Universal Robots PolyScope program: demo07_client_server.urp

Program demo07_client_server (installation=bbl_01 directory=/programs createdIn=5.7.0.90932 lastSavedIn=5.7.0.90932 robotSerialNumber=20205300236)
Calibrated DH parameters: a=[-0.000056, -0.241378, -0.055128, 0.000067, -0.000138, 0]; d=[0.151803, -14.462882, 131.163662, -116.569967, 0.085381, 0.091498]; alpha=[1.571556, -0.002127, 0.001765, 1.572165, -1.572257, 0]; deltaTheta=[0, 0.126747, 1.182538, -1.309285, 0, -0.000001]
BeforeStart
  Script: socket_close()
  Wait Sleep waitTime=0.25
  socket_is_open := False
  command_index := 0
Robot Program (runOnlyOnce=false)
  command_index := command_index+1
  Loop While (checkContinuously=false) expression=socket_is_open ≟  False
    socket_is_open := socket_open("192.168.1.1", 30000)
    Wait Sleep waitTime=0.5
  command := socket_read_ascii_float(5)
  response := "Unknown command"
  If command[0]≟5
    Switch expression=command[1]
      Case (caseValue=1)
        MoveL speed 250 mm/s, acceleration 1200 mm/s^2 (useActiveTCP=true) feature=Base
          Waypoint up_pose: TCP in base x=-233.309 y=250.262 z=151.642 mm, rx=0 ry=0 rz=0.7204 rad; joints [-69.689, -85.83, 83.489, -87.743, -89.951, 159.174] deg; TCP offset x=0 y=0 z=160 mm, rx=0 ry=3.1416 rz=0 rad
        response := "moved up"
      Case (caseValue=2)
        MoveJ speed 60 deg/s, acceleration 80 deg/s^2 (useActiveTCP=true) feature=Base
          Waypoint start_pose: TCP in base x=-233.309 y=250.262 z=117.159 mm, rx=0 ry=0 rz=0.7204 rad; joints [-69.688, -85.502, 92.427, -97.009, -89.967, 159.179] deg
        response := "moved down"
      Case (caseValue=3)
        URCap Gripper (Robotiq_Grippers, Robotiq Inc.) dataModel(position=100.0, force=100.0, speed=100.0, positionInDouble=100.0, forceInDouble=100.0, speedInDouble=100.0, slaveIds=[9], blocking=true)
        response := "close"
      Case (caseValue=4)
        URCap Gripper (Robotiq_Grippers, Robotiq Inc.) dataModel(position=0.0, force=100.0, speed=100.0, positionInDouble=0.0, forceInDouble=100.0, speedInDouble=100.0, slaveIds=[9], blocking=true)
        response := "open"
      Case (caseValue=99)
        response := "exiting"
    Script: socket_send_line(response)
    If command[1]≟99
      Script: socket_close()
      Halt
